(* CoDeSys 2.3 export: FBSYSTEMTIME.EXP *)

(* POU FbSystemTime, ST *)
FUNCTION_BLOCK FbSystemTime
VAR_INPUT
END_VAR
VAR_OUTPUT
	iHours:INT;
	iMinutes:INT;
END_VAR
VAR
	SystemTime: SysTime64;
	Time_date: SystemTimeDate;
	TimeDate: CurTimeEx;
END_VAR
(* Haal de systeemtijd op *)
TimeDate(SystemTime:= SystemTime, TimeDate:= Time_date);

(* Sla uren en minuten apart op *)
iHours := Time_Date.Hour;
iMinutes := Time_date.Minute;
END_FUNCTION_BLOCK
